FUNCTION_BLOCK XTS_System
VAR_INPUT
{attribute 'pingroup' := 'Power'}
	bEnable					: BOOL := FALSE;	//Enable operation (power movers, group all ...)
{attribute 'pingroup' := 'Power'}
	bReset					: BOOL := FALSE;	//Reset all axis
{attribute 'pingroup' := 'Manual'}
	bManual					: BOOL;				//Manual operation mode for movers test with collision avoidance
{attribute 'pingroup' := 'Manual'}
	udiMoverSelection		: UDINT := 0;		//Mover ID to move in manual mode. If ID is equal to zero all movers are moved
{attribute 'pingroup' := 'Manual'}
	udiStationSelection		: UDINT := 0;		//Target Station ID for mover selected. If zero manual mode works with target position input
{attribute 'pingroup' := 'Manual'}
	udiStopPositionSelection: UDINT := 1;		//Target Stop Position 1, 2 or 3
{attribute 'pingroup' := 'Manual'}
	bJogForward				: BOOL;				//Jog Forward command for manual mode operation 0
{attribute 'pingroup' := 'Manual'}
	bJogBackwards			: BOOL;				//Jog Backwards command for manual mode operation 0
{attribute 'pingroup' := 'Manual'}
	bManualMove				: BOOL;				//Move selected mover to target position at target velocity in manual mode operation 1
{attribute 'pingroup' := 'Manual'}
	bTeachStation			: BOOL;				//During manual mode flag up of teach station set the stop position of station equal to act mover position
{attribute 'pingroup' := 'Automatic'}
	bAutomatic				: BOOL;				//Automatic operation using stations
{attribute 'pingroup' := 'Profile'}
	lrTargetPosition		: LREAL := 0.0;		//Target Position [mm]
{attribute 'pingroup' := 'Profile'}
	lrTargetVelocity		: LREAL := 500.0;	//Target Velocity [mm]
{attribute 'pingroup' := 'Configuration'}
	stCfg					: stXTSCfg;			//General Configuration
{attribute 'pingroup' := 'Profile'}
	Direction				: tc3_mc3definitions.MC_DIRECTION := tc3_mc3definitions.MC_DIRECTION.mcDirectionPositive;	//Movement Direction	
{attribute 'pingroup' := 'SubElements'}
	ax						: ARRAY [1..Tc3_XTS_Utility.TcIoXtsEnvironmentParameterList.MaxXtsMoversPerXpu] OF FB_Mover;	//Movers
{attribute 'pingroup' := 'SubElements'}
	gp						: FB_GroupCA; //Group CA
{attribute 'pingroup' := 'SubElements'}
	aStations				: ARRAY [1..Tc3_XTS_Utility.TcIoXtsEnvironmentParameterList.MaxXtsInfoStation] OF FB_Station; //Stations
END_VAR
VAR_OUTPUT
{attribute 'pingroup' := 'Status'}
	sLog			 			: STRING := 'Invalid';
{attribute 'pingroup' := 'Status'}
	bError			 			: BOOL;
{attribute 'pingroup' := 'Status'}
	bReadyForMotion 			: BOOL;
{attribute 'pingroup' := 'Status'}
	bEnabled					: BOOL;
{attribute 'pingroup' := 'Manual'}
	bInManual					: BOOL;
{attribute 'pingroup' := 'Manual'}
	bTeachDone					: BOOL;
{attribute 'pingroup' := 'Automatic'}
	bInAutomatic				: BOOL;
{attribute 'pingroup' := 'XPU'}
	bInitDone					: BOOL;
{attribute 'pingroup' := 'XPU'}
	bMover1DetectionValid 		: BOOL;
{attribute 'pingroup' := 'XPU'}
	iOperationMode 				: OperationMode;
{attribute 'pingroup' := 'XPU'}
	AreAllPositionValid 		: BOOL;
{attribute 'pingroup' := 'XPU'}
	DetectedMoverCount 			: UDINT;
{attribute 'pingroup' := 'XPU'}
	ExpectedMoverCount 			: UDINT;
{attribute 'pingroup' := 'XPU'}
	HasMoverIdDetectorError		: BOOL;
{attribute 'pingroup' := 'XPU'}
	IsMoverIdDetectorActive		: BOOL;
{attribute 'pingroup' := 'XPU'}
	IsMoverIsDetectionValid		: BOOL;
{attribute 'pingroup' := 'XPU'}
	TrackCount					: UDINT;	
{attribute 'pingroup' := 'XPU'}
	PartCount					: UDINT;				
{attribute 'pingroup' := 'XPU'}
	lrPart1Length 				: LREAL;
{attribute 'pingroup' := 'XPU'}
	udiNumMovers  				: UDINT;
{attribute 'pingroup' := 'XPU'}
	udiPart1NumModules			: UDINT;
{attribute 'pingroup' := 'XPU'}
	eMoverType					: Tc3_XTS_Utility.MoverType;
{attribute 'pingroup' := 'GROUP CA'}
	eGroupState					: MC_GROUP_STATE;
{attribute 'pingroup' := 'GROUP CA'}
	bAllMoversStandStill		: BOOL;	
END_VAR
VAR
	(* XPU *)
	//{attribute 'hide'} 
	fbXTSEnv		 		: FB_TcIoXtsEnvironment;
	//{attribute 'hide'} 
	IXPU			 		: I_TcIoXtsProcessingUnit;
	//{attribute 'hide'} 
	IPart1			 		: I_TcIoXtsXpuPart;
	//{attribute 'hide'} 
	fbInfoServer			: FB_TcIoXtsInfoServer;
	//{attribute 'hide'} 
	aInfoServerOids			: ARRAY [1..Tc3_XTS_Utility.TcIoXtsEnvironmentParameterList.MaxXtsInfoServer] OF Tc3_XTS_Utility.OTCID;
	//{attribute 'hide'} 
	aStationsOTCID			: ARRAY [1..Tc3_XTS_Utility.TcIoXtsEnvironmentParameterList.MaxXtsInfoStation] OF Tc3_XTS_Utility.OTCID;
	//{attribute 'hide'} 
	aMoversOids				: ARRAY [1..Tc3_XTS_Utility.TcIoXtsEnvironmentParameterList.MaxXtsMoversPerXpu] OF Tc3_XTS_Utility.OTCID;
	//{attribute 'hide'} 
	GroupCAOTCID			: ARRAY [1..Tc3_XTS_Utility.TcIoXtsEnvironmentParameterList.MaxXtsCaGroup] OF Tc3_XTS_Utility.OTCID;
END_VAR
VAR
	bXPUInitDone			: BOOL;
	stVisuStationsCfg 		: ARRAY [1..Tc3_XTS_Utility.TcIoXtsEnvironmentParameterList.MaxXtsInfoStation] OF stStationCfg;
	stCurrentCfg			: stXTSCfg;			//General Configuration
	udiFirstMover			: UDINT;
END_VAR
VAR
	//Visu
	iFrameSelection			: INT;
END_VAR


//Initialization
Init(); 

//Operation
IF bInitDone THEN
	//Enable System
	bEnabled := Enable(bEnable);
	bInManual:= Manual(bManual AND bInAutomatic = FALSE AND bEnabled);
	bInAutomatic := Automatic(bAutomatic AND bInManual = FALSE AND bEnabled);
END_IF
Reset(bReset AND bAllMoversStandStill);
IF udiNumMovers <> 0 THEN
	//Call sub fb's like group CA, movers...
	Childs();
	//Status
	bReadyForMotion := gp.bError = FALSE AND bEnabled;
	bError			:= gp.bError;
END_IF

METHOD PRIVATE Automatic : BOOL
VAR_INPUT
	bEnable : BOOL;
END_VAR
VAR_INST
	iState 		: INT;
	bAllDone 	: BOOL;
	i 			: UDINT;
	bBusy		: BOOL;
END_VAR

//Error managment
IF bError OR bReset AND iState <> 999 THEN iState := 999; END_IF

CASE iState OF
	
	0 : IF bEnable THEN 
			stCurrentCfg := stCfg;
			//Reset all command
			FOR i:= 1 TO udiNumMovers DO
				ax[i].clearCmd();
			END_FOR
			iState := iState + 1; 
			bBusy  := TRUE;
		END_IF
		
	1 : //ReConfigure Stations
		sLog := 'Auto: Configure stations';
		bAllDone := TRUE;
		FOR i:= 1 TO Tc3_XTS_Utility.TcIoXtsEnvironmentParameterList.MaxXtsInfoStation DO
			aStations[i](stCfg := stCfg.stStationsCfg[i], (*ax := ax,*) udiNumMovers := udiNumMovers, lrPartLength := lrPart1Length, bInvertPolarity := ax[1].bMoverInverted, ax := ax);
			IF Tc3_XTS_Utility.TcIoXtsEnvironmentParameterList.MaxXtsInfoStation > 0 AND Tc3_XTS_Utility.TcIoXtsEnvironmentParameterList.MaxXtsInfoServer > 0 THEN  
				IF aStationsOTCID[i] <> 0 THEN
					bAllDone := bAllDone AND aStations[i].SetStationInfo(TRUE, OTCID := aStationsOTCID[i], i > stCurrentCfg.udiNumStations);
				END_IF
			ELSE
				bAllDone := TRUE;
			END_IF
			IF i<stCfg.udiNumStations THEN
					aStations[i].INextStation := aStations[i+1];	
			ELSIF i = stCfg.udiNumStations THEN	
					aStations[i].INextStation := aStations[1];	
			END_IF
		END_FOR
		IF bAllDone THEN
			//stVisuStationsCfg := stCfg.stStationsCfg;
			FOR i:= 1 TO Tc3_XTS_Utility.TcIoXtsEnvironmentParameterList.MaxXtsInfoStation DO
				IF Tc3_XTS_Utility.TcIoXtsEnvironmentParameterList.MaxXtsInfoStation > 0 AND Tc3_XTS_Utility.TcIoXtsEnvironmentParameterList.MaxXtsInfoServer > 0 THEN 
					aStations[i].SetStationInfo(FALSE, OTCID := aStationsOTCID[i], FALSE);
				END_IF
			END_FOR
			iState := iState + 1;
		END_IF

	2 : //Put all stations in auto mode
		sLog := 'Auto: Put stations in auto mode';
		bAllDOne := TRUE;
		FOR i:= 1 TO stCurrentCfg.udiNumStations DO
			bAllDone := bAllDOne AND aStations[i].Sequence2(TRUE, FALSE);
		END_FOR
		IF bAllDone THEN iState := iState + 1; END_IF
		IF bEnable = FALSE THEN iState := 100; END_IF
		
	3 : //Move all to zero position
		sLog := 'Auto: Move movers to start position';
		bAllDOne := FALSE;
		FOR i:= 1 TO udiNumMovers DO
			bAllDone := bAllDOne OR ax[i].moveca_gap(TRUE, 0.0, 1000.0, stCurrentCfg.lrMoverDistance);
		END_FOR
		IF bAllMoversStandStill AND bAllDone THEN
			udiFirstMover := WhoIsAtPos(0.0);
			FOR i:= 1 TO udiNumMovers DO
				ax[i].moveca(FALSE, 0.1, 0.0);
			END_FOR
			IF udiFirstMover <> 0 THEN
				iState := iState + 1;
			END_IF
		END_IF
		IF bEnable = FALSE THEN 
			iState := 100; 
		END_IF
		
	4 : //Gear in passive movers
		sLog := 'Auto: Gear in passive movers';
		bAllDone := TRUE;
		FOR i:= 1 TO udiNumMovers DO
			IF IsPassiveMover(i) THEN
				IF ax[1].bMoverInverted = FALSE THEN 
					bAllDone := bAllDone AND ax[i].gearIn(TRUE, 1, 1, ax[SEL(i = udiNumMovers, i+1, 1)].p_Axis);
				ELSE
					bAllDone := bAllDone AND ax[i].gearIn(TRUE, 1, 1, ax[SEL(i = 1, i-1, udiNumMovers)].p_Axis);
				END_IF
			END_IF
		END_FOR
		IF bAllDone THEN
			FOR i:= 1 TO udiNumMovers DO
				IF IsPassiveMover(i) THEN
					bAllDone := bAllDone AND ax[i].gearIn(FALSE, 1, 1, ax[SEL(i = udiNumMovers, i+1, 1)].p_Axis);
				END_IF
			END_FOR
			iState := iState + 1;
		END_IF

	5 :  //Add Movers to first station
		sLog := 'Auto: Add Movers to first station';
		FOR i:= 1 TO udiNumMovers DO
			IF IsPassiveMover(i) = FALSE THEN
				aStations[1].AddMover(ax[i].udiID);				
			END_IF
		END_FOR
		iState := iState + 1;
	
	6 : //Call stations auto mode
		sLog := CONCAT('Auto: Running ', INT_TO_STRING(iState));
		bAllDOne := TRUE;
		FOR i:= 1 TO stCurrentCfg.udiNumStations DO
			bAllDone := bAllDOne AND aStations[i].Sequence2(TRUE, FALSE);
		END_FOR
		IF bEnable = FALSE THEN 
			iState := 100; 
		END_IF
	
	100 : //Stop
		bAllDOne := TRUE;
		FOR i:= 1 TO stCurrentCfg.udiNumStations DO
			bAllDone := bAllDOne AND NOT aStations[i].Sequence2(FALSE, FALSE);
		END_FOR
		IF bAllDone THEN
			iState := iState + 1;
		END_IF
		
	101 : //Check for all StandStill
		bAllDone := TRUE;
		FOR i := 1 TO udiNumMovers DO
			bAllDone := bAllDone AND ax[i].standstill();
		END_FOR
		IF bAllDOne THEN
			iState := iState + 1;
		END_IF
		
	102 : //Gear Out
		bAllDone := TRUE;
		FOR i := 1 TO udiNumMovers DO
			IF IsPassiveMover(i) THEN
				bAllDone := bAllDone AND ax[i].gearOut(TRUE);
			END_IF
		END_FOR
		IF bAllDOne THEN
			FOR i := 1 TO udiNumMovers DO
				IF IsPassiveMover(i) THEN
					ax[i].gearOut(FALSE);
				END_IF
			END_FOR
			iState := iState + 1;
		END_IF
		
	103 : bBusy := FALSE;
		IF bEnable = FALSE THEN
			iState := 0;
		END_IF
		
	999 : //Error State 
		bBusy := FALSE;
		sLog := 'Auto: Abort'; 
		FOR i:=1 TO stCurrentCfg.udiNumStations DO
			//Abort Station Sequence
			aStations[i].Sequence2(FALSE, TRUE);
		END_FOR
		IF bEnable = FALSE THEN
			iState := 0;
		END_IF
		
END_CASE
Automatic := bBusy;
END_METHOD

METHOD PRIVATE Childs : BOOL
VAR_INPUT
END_VAR
VAR_INST
	i 	: UDINT;
	bAllDone : BOOL;
END_VAR
//Call Group CA
gp(ax:= ax, eGroupState=> eGroupState, bAllStandStill=> bAllMoversStandStill, bError=> );
//Call Movers
FOR i := 1 TO udiNumMovers DO
	ax[i]((*aStations := aStations,*) udiID=> );
END_FOR
//Call Stations
FOR i:= 1 TO stCfg.udiNumStations DO
	aStations[i](ax := ax);
END_FOR
END_METHOD

METHOD PRIVATE Enable : BOOL
VAR_INPUT
	bEnable		: BOOL;
END_VAR
VAR_INST
	iState 		: INT;
	bAllDone 	: BOOL;
	i 			: UDINT;
	bDone		: BOOL;
END_VAR

CASE iState OF
	
	0 : 
		IF bEnable THEN 
			FOR i := 1 TO udiNumMovers DO
				ax[i].ClearCmd();
			END_FOR
			gp.clearcmd();
			bDone := FALSE;
			iState := iState + 10; 
		END_IF
	
	10 : //Reset Movers
		sLog := 'Enable: Reset movers';
		bAllDone := TRUE;
		FOR i := 1 TO udiNumMovers DO
			bAllDone := bAllDone AND ax[i].reset(TRUE);
		END_FOR
		IF bAllDone THEN
			iState := iState + 1;
		END_IF
		
	11 : //Configure movers inversion
		sLog := 'Init: Configure movers inversion';
		bAllDone := TRUE;
		FOR i := 1 TO udiNumMovers DO
			bAllDone := bAllDone AND ax[i].InvertPolarity(TRUE, stCfg.bInvertPolarity);
		END_FOR
	 	IF bAllDOne THEN
			 FOR i := 1 TO udiNumMovers DO
			 	ax[i].InvertPolarity(FALSE, stCfg.bInvertPolarity);
		 	 END_FOR
			 iState := 20;
	 	END_IF
		
	20 : //Power all Axis
		sLog := 'Enable: Power on movers';
		bAllDone := TRUE;
		FOR i := 1 TO udiNumMovers DO
			bAllDone := bAllDone AND ax[i].power_on();
		END_FOR
		IF bAllDone THEN
			iState := iState + 1;
		END_IF
		
	21 : //Decopule axis
		sLog := 'Enable: Gear out movers';
		FOR i:=1 TO udiNumMovers DO
			IF ax[i].p_Axis.Status.Coupled  THEN
				//
				bAllDone := bAllDOne AND ax[i].gearOut(TRUE);
			END_IF
		END_FOR
		IF bAllDOne THEN
			FOR i:=1 TO udiNumMovers DO
				ax[i].gearOut(FALSE);
			END_FOR
			iState := 30;
		END_IF
		
	30 : //Reset Group
		sLog := 'Enable: Reset group CA';
		IF gp.reset(TRUE) THEN
			iState := iState + 10;
		END_IF
		
	40 : //Add all axis to group
		sLog := 'Enable: Add movers to group';
		bAllDone := TRUE;
		FOR i := 1 TO udiNumMovers DO
			bAllDone := bAllDone AND ax[i].add2Group(TRUE, ag := gp.ag);
		END_FOR
		IF bAllDone THEN
			FOR i := 1 TO udiNumMovers DO
				ax[i].add2Group(FALSE, ag := gp.ag);
			END_FOR
			iState := iState + 10;
		END_IF
		
	50 : //Enable group
		sLog := 'Enable: Enable group CA';
		IF gp.enable(TRUE) THEN
			iState := iState + 10;
		END_IF
		
	60 : //Jog Done
		sLog := 'Enable: Done!';
		 bDone := TRUE;
		 IF bEnable = FALSE THEN iState := 70; END_IF 

	70 : //Halt group
		sLog := 'Disable: Halt movers';
		bAllDone := TRUE;
		FOR i := 1 TO udiNumMovers DO
			bAllDone := bAllDone AND ax[i].haltca(TRUE);
		END_FOR
		IF bAllDone THEN
			iState := iState + 10;
		END_IF
		
	80 : //Disable
		sLog := 'Disable: Disable group CA';
		IF gp.disable(TRUE) THEN
			iState := iState + 10;
		END_IF		

	90 : //UnGroup
		sLog := 'Disable: UnGroup all movers';
		IF gp.ungroupall(TRUE) THEN
			iState := iState + 10;
		END_IF
	
	100 : //Power off all
		sLog := 'Disable: Power off all movers';
		bAllDone := TRUE;
		FOR i := 1 TO udiNumMovers DO
			bAllDone := bAllDone AND ax[i].power_off();
		END_FOR
		IF bAllDone THEN
			sLog := 'Disable: Done!';
			bDone := FALSE;
			iState := 0;
		END_IF
		 
END_CASE
Enable := bDone;
END_METHOD

METHOD PRIVATE Init
VAR_INST
	iState 		: INT;
	bAllDone 	: BOOL;
	i 			: UDINT;
END_VAR

//XPU Initialization
IF bXPUInitDone = FALSE THEN
	sLog := 'Init: Initialazing XPU';
	IF fbXTSEnv.Init(TRUE) THEN
		sLog := 'Init: XPU Initialazed';
		fbXTSEnv.Init(FALSE);
		bXPUInitDone := TRUE;
	END_IF	
END_IF

CASE iState OF
	
	0 : 
		IF bXPUInitDone THEN iState := iState + 10; END_IF
	
	10 : //Get XPU Parameters
		sLog := 'Init: Checking XPU parameters';
		Ixpu 						:= fbXTSEnv.XpuTcIo(1);
		IPart1						:= Ixpu.PartTcIo(1);
		iOperationMode 				:= Ixpu.GetOperationMode();
		AreAllPositionValid 		:= Ixpu.GetAreAllPositionsValid();
		DetectedMoverCount 			:= Ixpu.GetDetectedMoverCount();
		ExpectedMoverCount 			:= Ixpu.GetExpectedMoverCount();
		HasMoverIDDetectorError 	:= Ixpu.GetHasMoverIdDetectionError();
		IsMoveriddetectoractive 	:= Ixpu.GetIsMoverIdDetectionActive();
		ismoverisdetectionvalid 	:= Ixpu.GetIsMoverIdDetectionValid();
		TrackCount					:= Ixpu.GetTrackCount();
		PartCount					:= Ixpu.GetPartCount();
		lrPart1Length 				:= IPart1.GetLength();
		udiPart1NumModules			:= IPart1.GetModuleCount();
		udiNumMovers 				:= Ixpu.GetMoverCount();
		eMoverType					:= Ixpu.GetMoverType();
		
		IF (Ixpu.GetDetectedMoverCount() = Ixpu.GetExpectedMoverCount()) AND Ixpu.GetAreAllPositionsValid() THEN
			iState := iState + 10; 			
		END_IF

	20 : //Detect Mover 1 
		sLog := 'Init: Detecting mover 1';
		IF Ixpu.GetIsMoverIdDetectionValid() = FALSE THEN
			IF Ixpu.GetMoverIdDetectionMode() = 1 THEN
				Ixpu.TriggerMoverIdDetection();
				iState := iState + 1;
			ELSE
				bMover1DetectionValid := TRUE;
				iState := iState + 10;
			END_IF
		ELSE
			bMover1DetectionValid := TRUE;
			iState := iState + 10;
		END_IF
		
	21 : //Check Mover 1 Detection Valid
		IF Ixpu.GetIsMoverIdDetectionValid() THEN
			bMover1DetectionValid := TRUE;
			iState := 30;
		END_IF
	
	30 : //Get OIDS of Group CA
		sLog := 'Init: Getting group CA Oids';
		IF fbXTSEnv.GetCaGroupOids(TRUE) THEN
			fbXTSEnv.GetCaGroupOids(FALSE);
			GroupCAOTCID := fbXTSEnv.P_CaGroupOids;
			gp.fbXPUGroupCA.Init(FALSE, GroupCAOTCID[1]);
			iState := 31;
		END_IF
		
	31 : //Reset Group
		sLog := 'Init: Reset group CA';
		IF gp.reset(TRUE) THEN
			gp.reset(FALSE);
			iState := iState + 1;
		END_IF
		
	32 : //Disable Group in order to configure the Rail Length
		sLog := 'Init: UnGroup all';
		IF gp.ungroupall(TRUE) THEN
			gp.ungroupall(FALSE);
			iState := iState + 1;
		END_IF
		
	33 : //Set Group CA Rail Length equal to Part 1 length
		sLog := 'Init: Get group CA Oids';
		IF gp.fbXPUGroupCA.Init(TRUE, GroupCAOTCID[1]) THEN
			IF gp.fbXPUGroupCA.SetRailLength(lrPart1Length) THEN
				gp.fbXPUGroupCA.Init(FALSE, GroupCAOTCID[1]);
				iState := 40;		
			END_IF
		END_IF
		
	40 : //Get Info Server OIDS
		sLog := 'Init: Get Info Server Oids';
		IF Tc3_XTS_Utility.TcIoXtsEnvironmentParameterList.MaxXtsInfoServer > 0 THEN 
			IF fbXTSEnv.GetInfoServerOids(TRUE) THEN
				fbXTSEnv.GetInfoServerOids(FALSE);
				aInfoServerOids := fbXTSEnv.P_InfoServerOids;
				i:=1;
				fbInfoServer.Init(FALSE, aInfoServerOids[i]);
				iState := iState + 1;
			END_IF
		ELSE
			iState := iState + 10;
		END_IF

	41 : //Get OCID of Stations
		sLog := 'Init: Get Info Stations Oids';
		IF fbInfoServer.Init(TRUE, aInfoServerOids[i]) THEN
			IF fbInfoServer.GetInfoStationOids() THEN
				aStationsOTCID := fbInfoServer.P_InfoStationOids;
				fbInfoServer.Init(FALSE, aInfoServerOids[i]);
				FOR i:= 1 TO stCfg.udiNumStations DO
					aStations[i].SetStationInfo(FALSE, OTCID := aStationsOTCID[i], FALSE);
				END_FOR
				iState := 50;
			END_IF
		END_IF
		
	50 : //Get Mover OIDS
		sLog := 'Init: Get movers Oids';
		IF IXPU.GetMoverOids() THEN
			aMoversOids := IXPU.P_MoverOids;
			iState := iState + 1;
		END_IF
		
	51 : //Gear out movers
		sLog := 'Init: Gear out movers';
		bAllDone := TRUE;
		FOR i:=1 TO udiNumMovers DO
			IF ax[i].p_Axis.Status.Coupled THEN
				//
				bAllDone := bAllDOne AND ax[i].gearOut(TRUE);
			END_IF
		END_FOR
		IF bAllDOne THEN
			FOR i:=1 TO udiNumMovers DO
				ax[i].gearOut(FALSE);
			END_FOR
			iState := iState + 1;
		END_IF
		
	52 : //Reset Movers
		sLog := 'Init: Reset movers';
		bAllDOne := TRUE;
		 FOR i := 1 TO udiNumMovers DO
			 bAllDone := bAllDone AND ax[i].reset(TRUE);
		 END_FOR
		 IF bAllDOne THEN
			 FOR i := 1 TO udiNumMovers DO
			 	ax[i].reset(FALSE);
		 	 END_FOR
			 iState := iState + 1;
		 END_IF
		 
	53 : //Power off Movers
		sLog := 'Init: Power off movers';
		bAllDOne := TRUE;
		 FOR i := 1 TO udiNumMovers DO
			 bAllDone := bAllDone AND ax[i].power_off();
		 END_FOR
		 IF bAllDOne THEN
			 iState := iState + 1;
		 END_IF
		 
	54 : //Configure Movers
		sLog := 'Init: Configure movers';
		 bAllDone := TRUE;
		 FOR i := 1 TO udiNumMovers DO
			 bAllDone := bAllDone AND ax[i].InvertPolarity(TRUE, stCfg.bInvertPolarity);
		 END_FOR
	 	IF bAllDOne THEN
			 FOR i := 1 TO udiNumMovers DO
			 	ax[i].InvertPolarity(FALSE, stCfg.bInvertPolarity);
		 	 END_FOR
			 iState := 60;
	 	END_IF
		
	60 : //Set Stations configuration
		sLog := 'Init: Configure stations';
		bAllDone := TRUE;
		FOR i:= 1 TO Tc3_XTS_Utility.TcIoXtsEnvironmentParameterList.MaxXtsInfoStation DO
			aStations[i](stCfg := stCfg.stStationsCfg[i], (*ax := ax,*) udiNumMovers := udiNumMovers, lrPartLength := lrPart1Length, bInvertPolarity := ax[1].bMoverInverted, ax := ax);
			IF Tc3_XTS_Utility.TcIoXtsEnvironmentParameterList.MaxXtsInfoStation > 0 AND Tc3_XTS_Utility.TcIoXtsEnvironmentParameterList.MaxXtsInfoServer > 0 THEN  
				IF aStationsOTCID[i] <> 0 THEN
					bAllDone := bAllDone AND aStations[i].SetStationInfo(TRUE, OTCID := aStationsOTCID[i], i > stCfg.udiNumStations);
				END_IF
			ELSE
				bAllDone := TRUE;
			END_IF
			IF i<stCfg.udiNumStations THEN
					aStations[i].INextStation := aStations[i+1];	
			ELSIF i = stCfg.udiNumStations THEN	
					aStations[i].INextStation := aStations[1];	
			END_IF
		END_FOR
		IF bAllDone THEN
			stVisuStationsCfg := stCfg.stStationsCfg;
			FOR i:= 1 TO Tc3_XTS_Utility.TcIoXtsEnvironmentParameterList.MaxXtsInfoStation DO
				IF Tc3_XTS_Utility.TcIoXtsEnvironmentParameterList.MaxXtsInfoStation > 0 AND Tc3_XTS_Utility.TcIoXtsEnvironmentParameterList.MaxXtsInfoServer > 0 THEN 
					aStations[i].SetStationInfo(FALSE, OTCID := aStationsOTCID[i], FALSE);
				END_IF
			END_FOR
			iState := iState + 10;
		END_IF
		
	70 : //Jog Done
		 sLog := 'Init: Done!';
		 bInitDone 	:= TRUE;
		 iState := 71;
		 
	71 :
		//
			 
END_CASE
END_METHOD

METHOD IsPassiveMover : BOOL
VAR_INPUT
	ID 				: UDINT;
END_VAR
VAR_INST
	i 				: DINT;
	bFirstMoverEven : BOOL;
	iTmp			: udint;
END_VAR
IF stCFg.udiMoverMode = 2 THEN
	bFirstMoverEven := (udiFirstMover MOD 2) = 0;
	IsPassiveMover := ((ID MOD 2) <> 0 AND bFirstMoverEven) OR ((ID MOD 2) = 0 AND bFirstMoverEven = FALSE);
ELSIF stCFg.udiMoverMode = 3 THEN
	iTmp := udiFirstMover MOD 3;
	IsPassiveMover := ((ID MOD 3) <> iTmp); //AND bFirstMoverEven) OR ((ID MOD 3) <> 0 AND bFirstMoverEven = FALSE);
END_IF

	(*i := udiFirstMover-1;
	WHILE i = udiFirstMover+1 DO
		//
		IF ID = DINT_TO_UDINT(i) THEN 
			m_isPassiveMover := TRUE; 
			RETURN;
		END_IF
		i := i - 2;
		IF i < 1 THEN i := stCfg.uiTotalAxis; END_IF
	END_WHILE*)

	(*FOR i := udiFirstMover-1 TO 1 BY -2 DO
		IF ID = DINT_TO_UDINT(i) THEN 
			m_isPassiveMover := TRUE; 
			RETURN;
		END_IF	
		IF i < 1 THEN
			RETURN;
		END_IF
	END_FOR	
	
	FOR i := stCfg.uiTotalAxis TO udiFirstMover BY -2 DO
		IF ID = DINT_TO_UDINT(i) THEN 
			m_isPassiveMover := TRUE; 
			RETURN;
		END_IF	
		IF i < 1 THEN
			RETURN;
		END_IF
	END_FOR*)

//END_IF
END_METHOD

METHOD PRIVATE Manual : BOOL
VAR_INPUT
	bEnable 			: BOOL;
END_VAR
VAR_INST
	iState 				: INT;
	bAllDone 			: BOOL;
	i 					: UDINT;
	bBusy				: BOOL;
	fbRTRIG				: R_Trig;
	m_udiStationSelection : UDINT;
END_VAR

CASE iState OF
	0 : IF bEnable THEN 
			iState := iState + 1; 
			bBusy  := TRUE;
		END_IF
		
	1 : //Idle
		IF bEnable = FALSE THEN
			iState := 100;
		ELSIF bJogBackwards OR bJogForward THEN
			iState := 10; 
		ELSIF bManualMove AND udiStationSelection = 0 THEN
			//Move All with Target Position
			iState := 50; 
		ELSIF bManualMove AND udiStationSelection > 0 AND udiStationSelection < stCfg.udiNumStations+1 AND udiStopPositionSelection > 0 AND udiStopPositionSelection < 4 THEN
			//Move Mover to Station 
			iState := 60;
		ELSIF bTeachStation AND udiStationSelection > 0 AND udiMoverSelection > 0 AND udiStopPositionSelection > 0 AND udiStopPositionSelection < 4 THEN
			m_udiStationSelection := udiStationSelection;
			iState := 70;
		END_IF
		
	10 : //Manual mode operation 0 
		IF udiMoverSelection = 0 THEN
			bAllDone := TRUE;
			FOR i := 1 TO udiNumMovers DO
				bAllDone := bAllDone AND ax[i].jogca_velo(bJogBackwards, bJogForward, lrTargetVelocity) = FALSE;
			END_FOR
			IF bJogBackwards = FALSE AND bJogForward = FALSE AND bAllDone THEN
				iState := 1;
			END_IF	
		ELSE
			IF udiMoverSelection < 1 OR udiMoverSelection > udiNumMovers THEN udiMoverSelection := 1; END_IF
			IF ax[udiMoverSelection].jogca_velo(bJogBackwards, bJogForward, lrTargetVelocity) = FALSE AND bJogBackwards = FALSE AND bJogForward = FALSE THEN
				iState := 1;	
			END_IF
		END_IF
		
	50 : //Manual Operation with Target Position
		IF udiMoverSelection = 0 THEN
			FOR i := 1 TO udiNumMovers DO
				ax[i].moveca_direction(bManualMove, lrTargetPosition, lrTargetVelocity, Direction);
			END_FOR
			IF bAllMoversStandStill AND bManualMove = FALSE THEN
				iState := 1;
			END_IF
		ELSE ax[udiMoverSelection].moveca_direction(bManualMove, lrTargetPosition, lrTargetVelocity, Direction);
			IF bAllMoversStandStill AND bManualMove = FALSE THEN
				iState := 1;
			END_IF
		END_IF
		
	60 : //Manual Operation with Stations
		IF udiMoverSelection = 0 THEN
			FOR i := 1 TO udiNumMovers DO
				ax[i].moveca_direction(bManualMove, aStations[udiStationSelection].stCfg.lrStopPosition[udiStopPositionSelection] + aStations[udiStationSelection].stCfg.lrStartPosition, lrTargetVelocity, Direction);
			END_FOR
			IF bAllMoversStandStill AND bManualMove = FALSE THEN
				iState := 1;
			END_IF
		ELSE ax[udiMoverSelection].moveca_direction(bManualMove, aStations[udiStationSelection].stCfg.lrStopPosition[udiStopPositionSelection] + aStations[udiStationSelection].stCfg.lrStartPosition, lrTargetVelocity, Direction);
			IF bAllMoversStandStill AND bManualMove = FALSE THEN
				iState := 1;
			END_IF
		END_IF
		
	70 : //Teach Station
		stCfg.stStationsCfg[m_udiStationSelection].lrStopPosition[udiStopPositionSelection] := ax[udiMoverSelection].p_Axis.NcToPlc.ModuloSetPos-stCfg.stStationsCfg[m_udiStationSelection].lrStartPosition;
		bAllDone := TRUE;	
		FOR i:= 1 TO stCfg.udiNumStations DO
			bAllDone := bAllDone AND aStations[i].SetStationInfo(TRUE, OTCID := aStationsOTCID[i], FALSE);
		END_FOR
		IF bAllDone THEN
			FOR i:= 1 TO stCfg.udiNumStations DO
				aStations[i].SetStationInfo(FALSE, OTCID := aStationsOTCID[i], FALSE);
			END_FOR
			iState := iState + 1;
		END_IF
		
	71 : //Apply New Configuration
		bTeachDone := TRUE;
		IF bTeachStation = FALSE THEN
			bTeachDone := FALSE;
			iState := 1;
		END_IF
		
	100 : 
		bBusy := FALSE;
		iState := 0;
		
END_CASE
Manual := bBusy;
END_METHOD

METHOD Reset : BOOL
VAR_INPUT
	bEnable 	: BOOL;
END_VAR
VAR_INST
	iState		: INT;
	i 			: UDINT;
	bAllDOne 	: BOOL;
END_VAR

IF bEnable = FALSE THEN iState := 0; END_IF

CASE iState OF
	0 : IF bEnable THEN 
			FOR i:=1 TO udiNumMovers DO
				ax[i].reset(FALSE);
				ax[i].gearOut(FALSE);
			END_FOR
			gp.reset(FALSE);
			iState := iState + 1; 
		END_IF
	1 :
		bAllDone := TRUE;
		FOR i:=1 TO udiNumMovers DO
			IF udiFirstMover = 0 OR IsPassiveMover(i) = FALSE THEN
				bAllDone := bAllDOne AND ax[i].reset(TRUE);
			END_IF
		END_FOR
		IF bAllDone THEN
			FOR i:=1 TO udiNumMovers DO
				bAllDone := bAllDOne AND ax[i].reset(FALSE);
			END_FOR
			iState := iState + 1;
		END_IF
		
	2 : //Check if there is some axis coupled and decoupled (Is not possible to perform a reset group with axis coupled)
		bAllDone := TRUE;
		FOR i:=1 TO udiNumMovers DO
			IF ax[i].p_Axis.Status.Coupled  THEN
				//
				bAllDone := bAllDOne AND ax[i].gearOut(TRUE);
			END_IF
		END_FOR
		IF bAllDOne THEN
			FOR i:=1 TO udiNumMovers DO
				ax[i].gearOut(FALSE);
			END_FOR
			iState := iState + 1;
		END_IF
	
	3 : //Reset Group
		IF gp.reset(TRUE) THEN
			iState := iState + 1;
			gp.reset(FALSE);
		END_IF
		
	4 : //Reset Done
		Reset := TRUE;
		IF bEnable = FALSE THEN
			iState := 0;
		END_IF
END_CASE
END_METHOD

METHOD WhoIsAtPos : UDINT
VAR_INPUT
	lrPosition : LREAL;
END_VAR
VAR_INST
	i 			: UDINT;
	lrDistance	: LREAL;
END_VAR
FOR i := 1 TO udiNumMovers DO
	lrDistance := lrPosition - ax[i].p_ModulePos;
	IF ABS(lrDistance) < 1.0 OR ABS(lrDistance - lrPart1Length) < 1.0 THEN
		WhoIsAtPos := ax[i].udiID;
	END_IF
END_FOR
END_METHOD

END_FUNCTION_BLOCK

(* stored: Version 1.1.0.1, ProductVersion 3.1.4024.11
   POU XTS_System: Id {5ae7c6ed-3ba0-43e2-9653-91dd93f1278b}, SpecialFunc None
   Folder Utilities: Id {28bd214e-36ee-4540-9db5-d878c1bab5e3}
   Method Automatic: Id {ebab7c66-0335-4ae9-8609-64912689cde4}
   Method Childs: Id {6938a0e7-78d0-4df3-b2ed-deb98037208e}
   Method Enable: Id {578eff18-54db-4044-88c4-275ff826915e}
   Method Init: Id {39a6ee40-aeb1-4582-9e00-e75616bfd396}
   Method IsPassiveMover: Id {9b58f478-1f08-40ed-9940-9ad1d8c68206}
   Method Manual: Id {da1fa912-79d7-445a-b8e4-8be7db44a6c0}
   Method Reset: Id {911d81c3-9cf5-43a5-b484-4c6e2c0cab05}
   Method WhoIsAtPos: Id {44b13db2-c515-40a5-8b3e-0612ab9a1e21} *)
